PROGRAM PRG_VLS_MOTION
VAR
	 // VLS Motor 1; upper slit blade
    {attribute 'pytmc' := '
        pv: PLC:VLS:MOT:01
        field: DESC VLS Upper Slit Blade
    '}
    M1: DUT_MotionStage;
    fbMotion1: FB_MotionStage;

	 // VLS Motor 2; lower slit blade
    {attribute 'pytmc' := '
        pv: PLC:VLS:MOT:02
        field: DESC VLS Lower Slit Blade
    '}
    M2: DUT_MotionStage;
    fbMotion2: FB_MotionStage;
	
	
	// VLS Motor 3; right slit blade
    {attribute 'pytmc' := '
        pv: PLC:VLS:MOT:03
        field: DESC VLS Right Slit Blade
    '}
    M3: DUT_MotionStage;
    fbMotion3: FB_MotionStage;
	
	// VLS Motor 4; left slit blade
    {attribute 'pytmc' := '
        pv: PLC:VLS:MOT:04
        field: DESC VLS Left Slit Blade
    '}
    M4: DUT_MotionStage;
    fbMotion4: FB_MotionStage;
	
	// VLS Motor 5; focusing mirror
    {attribute 'pytmc' := '
        pv: PLC:VLS:MOT:05
        field: DESC VLS Motor 5
    '}
    M5: DUT_MotionStage;
    fbMotion5: FB_MotionStage;
	
	// VLS Motor 6; grating
    {attribute 'pytmc' := '
        pv: PLC:VLS:MOT:06
        field: DESC VLS Motor 6
    '}
    M6: DUT_MotionStage;
    fbMotion6: FB_MotionStage;
	
	// VLS Motor 7; camera pitch
    {attribute 'pytmc' := '
        pv: PLC:VLS:MOT:07
        field: DESC VLS Motor 7
    '}
    M7: DUT_MotionStage;
    fbMotion7: FB_MotionStage;
	
	// VLS Motor 8; camera translation
    {attribute 'pytmc' := '
        pv: PLC:VLS:MOT:08
        field: DESC VLS Motor 8
    '}
    M8: DUT_MotionStage;
    fbMotion8: FB_MotionStage;
END_VAR

fbMotion1(stMotionStage := M1); // top slit blade
M1.bHardwareEnable := TRUE;
M1.bPowerSelf := TRUE;
M1.bLimitForwardEnable := M1.Axis.NcToPlc.ActPos < 18.8; // old limit 19
M1.bLimitBackwardEnable := M1.Axis.NcToPlc.ActPos > 0.2; // old limit 0

fbMotion2(stMotionStage := M2); // bottom slit blade
M2.bHardwareEnable := TRUE;
M2.bPowerSelf := TRUE;
M2.bLimitForwardEnable := M2.Axis.NcToPlc.ActPos < 23.8; // old limit 24
M2.bLimitBackwardEnable := M2.Axis.NcToPlc.ActPos > 0.2; // old limit 0

fbMotion3(stMotionStage := M3); // right slit blade
M3.bHardwareEnable := TRUE;
M3.bPowerSelf := TRUE;
M3.bLimitForwardEnable := M3.Axis.NcToPlc.ActPos < 47.9; // old limit 48.1
M3.bLimitBackwardEnable := M3.Axis.NcToPlc.ActPos > 0.2; // old limit 0

fbMotion4(stMotionStage := M4); // left slit blade
M4.bHardwareEnable := TRUE;
M4.bPowerSelf := TRUE;
M4.bLimitForwardEnable := M4.Axis.NcToPlc.ActPos < 48.8; // old limit 49
M4.bLimitBackwardEnable := M4.Axis.NcToPlc.ActPos > 0.2; // old limit 0

fbMotion5(stMotionStage := M5); // focusing mirror
M5.bHardwareEnable := TRUE;
M5.bPowerSelf := TRUE;
M5.bLimitForwardEnable := M5.Axis.NcToPlc.ActPos < 0.4; // old value 0.43
M5.bLimitBackwardEnable := M5.Axis.NcToPlc.ActPos > -3.4; // old value -3.47

fbMotion6(stMotionStage := M6); // grating
M6.bHardwareEnable := TRUE;
M6.bPowerSelf := TRUE;
M6.bLimitForwardEnable := M6.Axis.NcToPlc.ActPos < 1.0; // old value 1.2
M6.bLimitBackwardEnable := M6.Axis.NcToPlc.ActPos > -1.5; // old value -1.74

fbMotion7(stMotionStage := M7); // camera pitch
M7.bHardwareEnable := TRUE;
M7.bPowerSelf := TRUE;
M7.bLimitForwardEnable := M7.Axis.NcToPlc.ActPos < 1.0; // old value 1.2
M7.bLimitBackwardEnable := M7.Axis.NcToPlc.ActPos > -9.8; // old value -10

fbMotion8(stMotionStage := M8); // camera translation
M8.bHardwareEnable := TRUE;
M8.bPowerSelf := TRUE;
M8.bLimitForwardEnable := M8.Axis.NcToPlc.ActPos < 15.5; // old value 16
M8.bLimitBackwardEnable := M8.Axis.NcToPlc.ActPos > -15; // old value -15.5

END_PROGRAM

(* stored: Version 1.1.0.1, ProductVersion 3.1.4020.14
   POU PRG_VLS_MOTION: Id {f5736d79-b854-4294-93a7-0582bfcfe282}, SpecialFunc None *)
